// TIA Portal V20 export
TYPE "UDT_OPC_Button"
   STRUCT
      bBlink : Bool;
      bClick : Bool;
      bEnable : Bool;
      bIsPressed : Bool;
      eColor : Int;   // @Max:4
   END_STRUCT;
END_TYPE
